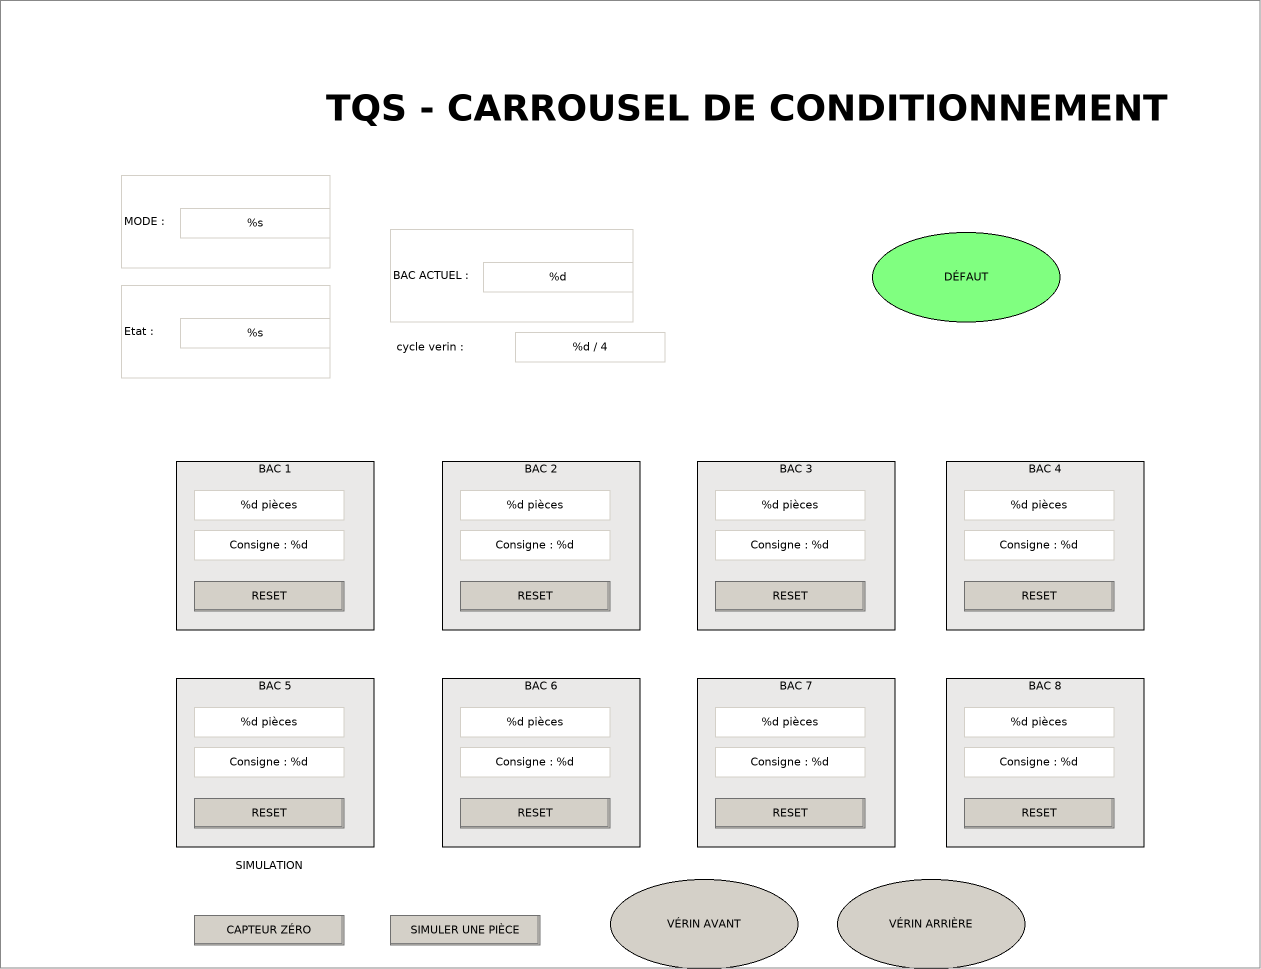
VISUALIZATION Visualization  // 1261x969
    Label (233,4 1028x208), "TQS - CARROUSEL DE CONDITIONNEMENT"
    Textfield (390,229 243x93), "BAC ACTUEL :"
    Textfield (483,262 150x30), "%d", text variable: MAIN.nBacOut
    Rectangle (176,461 198x169), "BAC 1", colour toggle: MAIN.aBacActifVisu[1]
    Button (194,581 150x30), "RESET"
        tap MAIN.aResetBacIn[1]
    Textfield (194,490 150x30), "%d pièces", text variable: MAIN.aPieceBacOut[1]
    Textfield (194,530 150x30), "Consigne : %d", text variable: MAIN.nPieceBacCmd
    Rectangle (442,461 198x169), "BAC 2", colour toggle: MAIN.aBacActifVisu[2]
    Button (460,581 150x30), "RESET"
        tap MAIN.aResetBacIn[2]
    Textfield (460,490 150x30), "%d pièces", text variable: MAIN.aPieceBacOut[2]
    Textfield (460,530 150x30), "Consigne : %d", text variable: MAIN.nPieceBacCmd
    Rectangle (697,461 198x169), "BAC 3", colour toggle: MAIN.aBacActifVisu[3]
    Button (715,581 150x30), "RESET"
        tap MAIN.aResetBacIn[3]
    Textfield (715,490 150x30), "%d pièces", text variable: MAIN.aPieceBacOut[3]
    Textfield (715,530 150x30), "Consigne : %d", text variable: MAIN.nPieceBacCmd
    Rectangle (176,678 198x169), "BAC 5", colour toggle: MAIN.aBacActifVisu[5]
    Button (194,798 150x30), "RESET"
        tap MAIN.aResetBacIn[5]
    Textfield (194,707 150x30), "%d pièces", text variable: MAIN.aPieceBacOut[5]
    Textfield (194,747 150x30), "Consigne : %d", text variable: MAIN.nPieceBacCmd
    Rectangle (442,678 198x169), "BAC 6", colour toggle: MAIN.aBacActifVisu[6]
    Button (460,798 150x30), "RESET"
        tap MAIN.aResetBacIn[6]
    Textfield (460,707 150x30), "%d pièces", text variable: MAIN.aPieceBacOut[6]
    Textfield (460,747 150x30), "Consigne : %d", text variable: MAIN.nPieceBacCmd
    Rectangle (697,678 198x169), "BAC 7", colour toggle: MAIN.aBacActifVisu[7]
    Button (715,798 150x30), "RESET"
        tap MAIN.aResetBacIn[7]
    Textfield (715,707 150x30), "%d pièces", text variable: MAIN.aPieceBacOut[7]
    Textfield (715,747 150x30), "Consigne : %d", text variable: MAIN.nPieceBacCmd
    Rectangle (946,461 198x169), "BAC 4", colour toggle: MAIN.aBacActifVisu[4]
    Button (964,581 150x30), "RESET"
        tap MAIN.aResetBacIn[4]
    Textfield (964,490 150x30), "%d pièces", text variable: MAIN.aPieceBacOut[4]
    Textfield (964,530 150x30), "Consigne : %d", text variable: MAIN.nPieceBacCmd
    Rectangle (946,678 198x169), "BAC 8", colour toggle: MAIN.aBacActifVisu[8]
    Button (964,798 150x30), "RESET"
        tap MAIN.aResetBacIn[8]
    Textfield (964,707 150x30), "%d pièces", text variable: MAIN.aPieceBacOut[8]
    Textfield (964,747 150x30), "Consigne : %d", text variable: MAIN.nPieceBacCmd
    Textfield (121,175 209x93), "MODE :"
    Textfield (180,208 150x30), "%s", text variable: MAIN.sModeVisu
    Textfield (121,285 209x93), "Etat :"
    Textfield (180,318 150x30), "%s", text variable: MAIN.sEtatCycleVisu
    Ellipse (872,232 188x90), "DÉFAUT", colour toggle: MAIN.bDefautOut
    Ellipse (610,879 188x90), "VÉRIN AVANT", colour toggle: MAIN.bVerinAvOut
    Ellipse (837,879 188x90), "VÉRIN ARRIÈRE", colour toggle: MAIN.bVerinArOut
    Textfield (515,332 150x30), "%d / 4", text variable: MAIN.nImpOut
    Label (355,332 150x30), "cycle verin :"
    Button (194,915 150x30), "CAPTEUR ZÉRO"
        toggle MAIN.bZeroIn
    Button (390,915 150x30), "SIMULER UNE PIÈCE"
        toggle MAIN.bLaserIn
    Label (194,857 150x30), "SIMULATION"
END_VISUALIZATION

(* stored: Version 1.1.0.1
   Visu Visualization: Id {c8bd2468-41a2-4718-b501-bdfb84a86044} *)
